SUBAPPLICATION GreenRedBackground_aux_AX (* Umschalten Hintergrundfarbe *)
  (* Standard: 61499-2; Description: Copyright (c) 2022 HR Agrartechnik GmbH This program and the accompanying materials are made available under the terms of the Eclipse Public License 2.0 which is available at https://www.eclipse.org/legal/epl-2.0/ SPDX-License-Identifier: EPL-2.0 *)
  (* Version 1.0, 2022-11-10, Franz Höpfinger, HR Agrartechnik GmbH *)
  PACKAGE MyLib::sys;
  IMPORT isobus::UT::Q::const::IDs::ID_NULL;
  IMPORT isobus::UT::Q::const::colours::COLOR_GREEN;
  IMPORT isobus::UT::Q::const::colours::COLOR_RED;
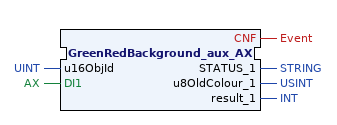
  EVENT_OUTPUT
    CNF; (* Execution Confirmation *)
  END_EVENT
  VAR_INPUT
    u16ObjId : UINT := ID_NULL; (* Object ID Softkey/Button *)
  END_VAR
  VAR_OUTPUT
    STATUS_1 : STRING; (* Service Status *)
    u8OldColour_1 : USINT; (* Old value of ID *)
    result_1 : INT; (* retval see description *)
  END_VAR
  SOCKETS
    DI1 : adapter::types::unidirectional::AX; (* Selector *)
  END_SOCKETS
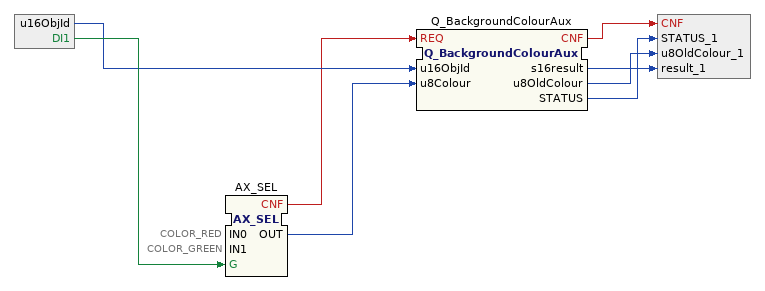
  FBS
    Q_BackgroundColourAux : isobus::UT::Q::Q_BackgroundColourAux;
    AX_SEL : adapter::iec61131::selection::AX_SEL(IN0 := COLOR_RED, IN1 := COLOR_GREEN);
  END_FBS
  EVENT_CONNECTIONS
    Q_BackgroundColourAux.CNF TO CNF;
    AX_SEL.CNF TO Q_BackgroundColourAux.REQ;
  END_CONNECTIONS
  DATA_CONNECTIONS
    u16ObjId TO Q_BackgroundColourAux.u16ObjId;
    Q_BackgroundColourAux.s16result TO result_1;
    Q_BackgroundColourAux.u8OldColour TO u8OldColour_1;
    Q_BackgroundColourAux.STATUS TO STATUS_1;
    AX_SEL.OUT TO Q_BackgroundColourAux.u8Colour;
  END_CONNECTIONS
  ADAPTER_CONNECTIONS
    DI1 TO AX_SEL.G;
  END_CONNECTIONS
END_SUBAPPLICATION
